TYPE DUT_SensorHGS:
STRUCT 
	fCntsInEGU:			REAL;
	sEGU:				STRING;
	sName:				STRING;
	fValue:				REAL;
	iRawCnts AT %I*:	DINT;
	iOffset:			DINT;
	q_iRawCnts AT %I*:	UINT;
END_STRUCT
END_TYPE

(* stored: Version 1.1.0.1, ProductVersion 3.1.4022.18
   DUT DUT_SensorHGS: Id {2917fbec-0023-49ad-b5e9-7d9d5133fd10} *)
